// TIA Portal V21 export
VAR_GLOBAL   // PLC tag table "BOMBA (BH-01B)"
END_VAR
